PROGRAM MAIN
VAR
	
	prox_sensors: ARRAY [1..8] OF BOOL;
	
END_VAR



prox_sensors := GVL_input.sensor;

END_PROGRAM

(* stored: Version 1.1.0.1, ProductVersion 3.1.4024.12
   POU MAIN: Id {66d06c91-d797-4675-9bef-0baaaa0a4f7b}, SpecialFunc None *)
